// TIA Portal V20 export
TYPE "typeCmControlNodeInterlock"
// stored: Namespace Unit1.Em6
   STRUCT
      visionUnit { ExternalWritable := 'False'} : "LER_typeAxisInterlock";
      visionPusherSupport { ExternalWritable := 'False'} : "LER_typeTwoWayActuatorInterlock";
   END_STRUCT;
END_TYPE
